// TIA Portal V15.1 export
// export: Created 2026-01-09T13:45:15.5623148Z, ExportSetting WithDefaults, WithReadOnly, DisplayName Totally Integrated Automation Portal, DisplayVersion V15.1 Update 8, DisplayName TIA Portal Openness, DisplayVersion V15.1 Update 8, DisplayName STEP 7 Professional, DisplayVersion V15.1 Update 8, DisplayName WinCC Advanced, DisplayVersion V15.1 Update 8
FUNCTION "FCXL_CCD_SB1" : Void   // FC17, LAD
{ S7_Optimized_Access := 'TRUE' }
VERSION : 0.1
// stored: AutoNumber true, CodeModifiedDate 2026-01-04T14:27:05.8156344Z, CompileDate 2026-01-04T14:27:05.8623022Z, CreationDate 2024-10-13T15:07:34.9617085Z, HandleErrorsWithinBlock false, InterfaceModifiedDate 2024-08-08T03:53:18.695573Z, IsConsistent true, IsIECCheckEnabled false, IsKnowHowProtected false, IsWriteProtected false, LibraryConformanceStatus Error: The block contains calls of single instances. Warning: The object contains access to global data blocks. Warning: The block contains direct access to inputs, outputs, bit memories, indirect access to the registry or indirect access to external memory areas that are unknown at the time of compilation., ModifiedDate 2026-01-04T14:27:05.8156344Z, ParameterModified 2024-08-08T03:53:18.695573Z, PLCSimAdvancedSupport false, SetENOAutomatically False, StructureModified 2024-08-08T03:53:18.695573Z, UDAEnableTagReadback false
   VAR_TEMP   // added for the SCL form of the ladder/FBD networks
      _w1 : Bool;
      _w2 : Bool;
      _w3 : Bool;
   END_VAR
BEGIN

REGION Network 1
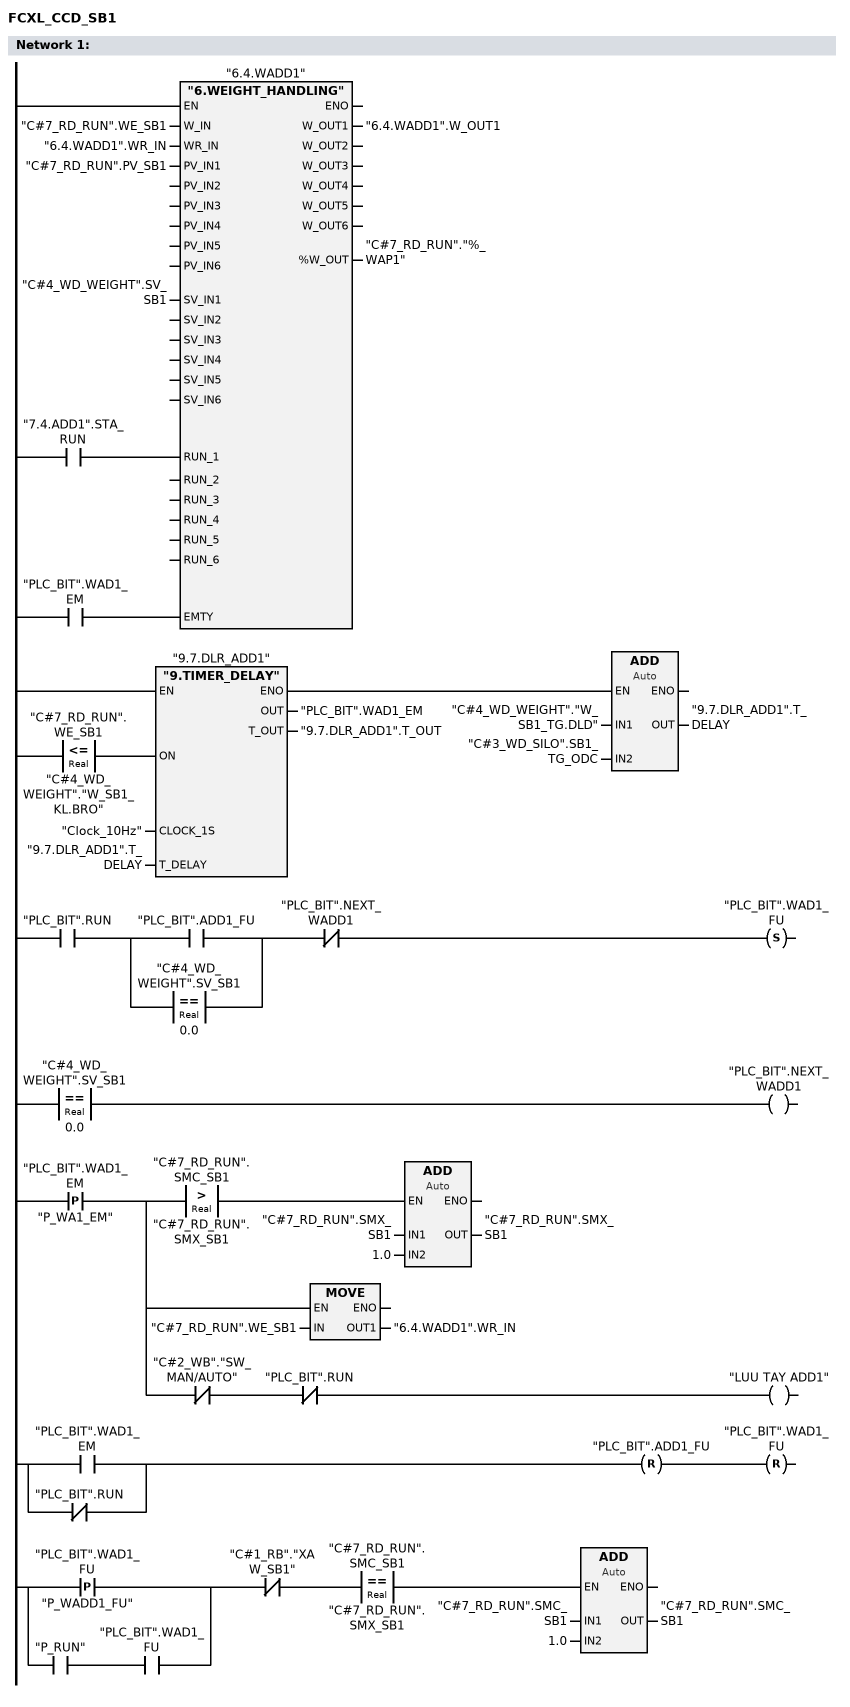
   RUNG wire#powerrail
      "6.4.WADD1"(RUN_1 := wire#w1, EMTY := wire#w2, W_IN := "C#7_RD_RUN".WE_SB1, WR_IN := "6.4.WADD1".WR_IN, PV_IN1 := "C#7_RD_RUN".PV_SB1, PV_IN2 :=, PV_IN3 :=, PV_IN4 :=, PV_IN5 :=, PV_IN6 :=, SV_IN1 := "C#4_WD_WEIGHT".SV_SB1, SV_IN2 :=, SV_IN3 :=, SV_IN4 :=, SV_IN5 :=, SV_IN6 :=, RUN_2 :=, RUN_3 :=, RUN_4 :=, RUN_5 :=, RUN_6 :=, W_OUT1 => "6.4.WADD1".W_OUT1, W_OUT2 =>, W_OUT3 =>, W_OUT4 =>, W_OUT5 =>, W_OUT6 =>, "%W_OUT" => "C#7_RD_RUN"."%_WAP1")
   END_RUNG
   RUNG wire#powerrail
      Contact( "7.4.ADD1".STA_RUN )
   END_RUNG wire#w1
   RUNG wire#powerrail
      Contact( "PLC_BIT".WAD1_EM )
   END_RUNG wire#w2
   RUNG wire#powerrail
      "9.7.DLR_ADD1"(ON := wire#w3, CLOCK_1S := "Clock_10Hz", T_DELAY := "9.7.DLR_ADD1".T_DELAY, OUT => "PLC_BIT".WAD1_EM, T_OUT => "9.7.DLR_ADD1".T_OUT)
      Add(in1 := "C#4_WD_WEIGHT"."W_SB1_TG.DLD", in2 := "C#3_WD_SILO".SB1_TG_ODC, out => "9.7.DLR_ADD1".T_DELAY)
   END_RUNG
   RUNG wire#powerrail
      { S7_Templates := "SrcType := Real" } LE_Contact(in1 := "C#7_RD_RUN".WE_SB1, in2 := "C#4_WD_WEIGHT"."W_SB1_KL.BRO")
   END_RUNG wire#w3
   RUNG wire#powerrail
      Contact( "PLC_BIT".RUN )
      wire#w4
      Contact( "PLC_BIT".ADD1_FU )
      wire#w5
      I_Contact( "PLC_BIT".NEXT_WADD1 )
      S_Coil( "PLC_BIT".WAD1_FU )
   END_RUNG
   RUNG wire#w4
      { S7_Templates := "SrcType := Real" } EQ_Contact(in1 := "C#4_WD_WEIGHT".SV_SB1, in2 := 0.0)
   END_RUNG wire#w5
   RUNG wire#powerrail
      { S7_Templates := "SrcType := Real" } EQ_Contact(in1 := "C#4_WD_WEIGHT".SV_SB1, in2 := 0.0)
      Coil( "PLC_BIT".NEXT_WADD1 )
   END_RUNG
   RUNG wire#powerrail
      P_Contact(operand := "PLC_BIT".WAD1_EM, bit := "P_WA1_EM")
      wire#w6
      { S7_Templates := "SrcType := Real" } GT_Contact(in1 := "C#7_RD_RUN".SMC_SB1, in2 := "C#7_RD_RUN".SMX_SB1)
      Add(in1 := "C#7_RD_RUN".SMX_SB1, in2 := 1.0, out => "C#7_RD_RUN".SMX_SB1)
   END_RUNG
   RUNG wire#w6
      Move(in := "C#7_RD_RUN".WE_SB1, out1 => "6.4.WADD1".WR_IN)
   END_RUNG
   RUNG wire#w6
      I_Contact( "C#2_WB"."SW_MAN/AUTO" )
      I_Contact( "PLC_BIT".RUN )
      Coil( "LUU TAY ADD1" )
   END_RUNG
   RUNG wire#powerrail
      Contact( "PLC_BIT".WAD1_EM )
      wire#w7
      R_Coil( "PLC_BIT".ADD1_FU )
      R_Coil( "PLC_BIT".WAD1_FU )
   END_RUNG
   RUNG wire#powerrail
      I_Contact( "PLC_BIT".RUN )
   END_RUNG wire#w7
   RUNG wire#powerrail
      P_Contact(operand := "PLC_BIT".WAD1_FU, bit := "P_WADD1_FU")
      wire#w8
      I_Contact( "C#1_RB"."XA W_SB1" )
      { S7_Templates := "SrcType := Real" } EQ_Contact(in1 := "C#7_RD_RUN".SMC_SB1, in2 := "C#7_RD_RUN".SMX_SB1)
      Add(in1 := "C#7_RD_RUN".SMC_SB1, in2 := 1.0, out => "C#7_RD_RUN".SMC_SB1)
   END_RUNG
   RUNG wire#powerrail
      Contact( "P_RUN" )
      Contact( "PLC_BIT".WAD1_FU )
   END_RUNG wire#w8
   // the same network as SCL:
   "6.4.WADD1"(W_IN := "C#7_RD_RUN".WE_SB1,   // "6.WEIGHT_HANDLING"
               WR_IN := "6.4.WADD1".WR_IN,
               PV_IN1 := "C#7_RD_RUN".PV_SB1,
               SV_IN1 := "C#4_WD_WEIGHT".SV_SB1,
               RUN_1 := "7.4.ADD1".STA_RUN,
               EMTY := "PLC_BIT".WAD1_EM,
               W_OUT1 => "6.4.WADD1".W_OUT1,
               "%W_OUT" => "C#7_RD_RUN"."%_WAP1");
   "9.7.DLR_ADD1"(ON := "C#7_RD_RUN".WE_SB1 <= "C#4_WD_WEIGHT"."W_SB1_KL.BRO",   // "9.TIMER_DELAY"
                  CLOCK_1S := "Clock_10Hz",
                  T_DELAY := "9.7.DLR_ADD1".T_DELAY,
                  OUT => "PLC_BIT".WAD1_EM,
                  T_OUT => "9.7.DLR_ADD1".T_OUT,
                  ENO => #_w1);
   IF #_w1 THEN "9.7.DLR_ADD1".T_DELAY := "C#4_WD_WEIGHT"."W_SB1_TG.DLD" + "C#3_WD_SILO".SB1_TG_ODC; END_IF;
   IF "PLC_BIT".RUN AND ("PLC_BIT".ADD1_FU OR ("C#4_WD_WEIGHT".SV_SB1 = 0.0)) AND NOT "PLC_BIT".NEXT_WADD1 THEN
       "PLC_BIT".WAD1_FU := TRUE;
   END_IF;
   "PLC_BIT".NEXT_WADD1 := "C#4_WD_WEIGHT".SV_SB1 = 0.0;
   #_w2 := "PLC_BIT".WAD1_EM AND NOT "P_WA1_EM";   // rising edge of "PLC_BIT".WAD1_EM
   "P_WA1_EM" := "PLC_BIT".WAD1_EM;
   IF #_w2 AND ("C#7_RD_RUN".SMC_SB1 > "C#7_RD_RUN".SMX_SB1) THEN
       "C#7_RD_RUN".SMX_SB1 := "C#7_RD_RUN".SMX_SB1 + 1.0;
   END_IF;
   IF #_w2 THEN "6.4.WADD1".WR_IN := "C#7_RD_RUN".WE_SB1; END_IF;
   "LUU TAY ADD1" := #_w2 AND NOT "C#2_WB"."SW_MAN/AUTO" AND NOT "PLC_BIT".RUN;
   IF "PLC_BIT".WAD1_EM OR NOT "PLC_BIT".RUN THEN
       "PLC_BIT".ADD1_FU := FALSE;
       "PLC_BIT".WAD1_FU := FALSE;
   END_IF;
   #_w3 := "PLC_BIT".WAD1_FU AND NOT "P_WADD1_FU";   // rising edge of "PLC_BIT".WAD1_FU
   "P_WADD1_FU" := "PLC_BIT".WAD1_FU;
   IF (#_w3 OR ("P_RUN" AND "PLC_BIT".WAD1_FU)) AND NOT "C#1_RB"."XA W_SB1" AND ("C#7_RD_RUN".SMC_SB1 = "C#7_RD_RUN".SMX_SB1) THEN
       "C#7_RD_RUN".SMC_SB1 := "C#7_RD_RUN".SMC_SB1 + 1.0;
   END_IF;
END_REGION
END_FUNCTION
